PROGRAM MAIN
VAR
END_VAR

P_Task1();

END_PROGRAM

(* stored: Version 1.1.0.1, ProductVersion 3.1.4024.12
   POU MAIN: Id {3f9925b0-dc3e-4f0c-8de8-e07bea341e3a}, SpecialFunc None *)
